// TwinCAT 3 PLC project Untitled1
// ProgramVersion: 3.1.4023.0
// libraries:
//   Tc2_Standard, * (Beckhoff Automation GmbH)
//   Tc2_System, * (Beckhoff Automation GmbH)
//   Tc3_Module, * (Beckhoff Automation GmbH)
// project tree:
//   / PlcTask.TcTTO
//   POUs/ MAIN.TcPOU
// real-time tasks:
//   TASK Task 1: cycle T#2ms, priority 2, ADS port 301
//   TASK PlcTask: cycle T#2ms, priority 1, ADS port 350

CONFIGURATION Untitled1
    RESOURCE PLC ON TwinCAT3
        TASK PlcTask(INTERVAL := T#2ms, PRIORITY := 1);
        PROGRAM MAIN WITH PlcTask : MAIN;
    END_RESOURCE
END_CONFIGURATION

// ---- POUs/MAIN.TcPOU
PROGRAM MAIN
VAR
    fbGetCurTaskIdx  : GETCURTASKINDEX;
    nCycleTime       : UDINT;
	fb_cpu_cnt		 : GETCPUACCOUNT; 
	start 			 : ULINT; // 100ns
	now				 : ULINT; // 100ns
	passed			 : ULINT; // 100ns
	b_initialized 	 : BOOL;	
	bExceed			 AT %I* : BOOL;
END_VAR

IF NOT b_initialized THEN
	b_initialized := TRUE;
	
	fbGetCurTaskIdx();
	nCycleTime := _TaskInfo[fbGetCurTaskIdx.index].CycleTime;
END_IF

IF bExceed THEN
	bExceed := FALSE;
	
	fb_cpu_cnt(cpuAccountDW =>start);

	REPEAT
		fb_cpu_cnt(cpuAccountDW =>now);
		passed := now - start;
	UNTIL
		passed > nCycleTime
		//passed +10000 > nCycleTime // >> High Load
	END_REPEAT
END_IF

END_PROGRAM
